// TIA Portal V16 export
// export: Created 2023-09-11T12:14:51.1549181Z, ExportSetting WithDefaults, DisplayName Totally Integrated Automation Portal, DisplayVersion V16 Update 6, DisplayName TIA Portal Version Control Interface, DisplayVersion V16 Update 2, DisplayName TIA Portal Openness, DisplayVersion V16 Update 6, DisplayName STEP 7 Professional, DisplayVersion V16 Update 6, DisplayName STEP 7 Safety, DisplayVersion V16, DisplayName WinCC Advanced, DisplayVersion V16 Update 6
ORGANIZATION_BLOCK "Cyclic interrupt"   // OB30, LAD, CyclicInterrupt
{ S7_Optimized_Access := 'TRUE' }
AUTHOR : RTecmer
VERSION : 0.1
// stored: AutoNumber true, IsIECCheckEnabled false, SetENOAutomatically false
   VAR_TEMP
      Temp_SV_Int : Int;
      PV_Temp : Real;
      Temp_1 : Real;
   END_VAR
   VAR_TEMP   // added for the SCL form of the ladder/FBD networks
      _w1 : Bool;
      _w2 : Bool;
   END_VAR
BEGIN

REGION Network 1: Wyłączenie wejścia pradowego w regulatorze PID
   // Przełączenie na Input PID  (wejście wartościci zadanej) wyłaczenie wejścia prądowego input_PER
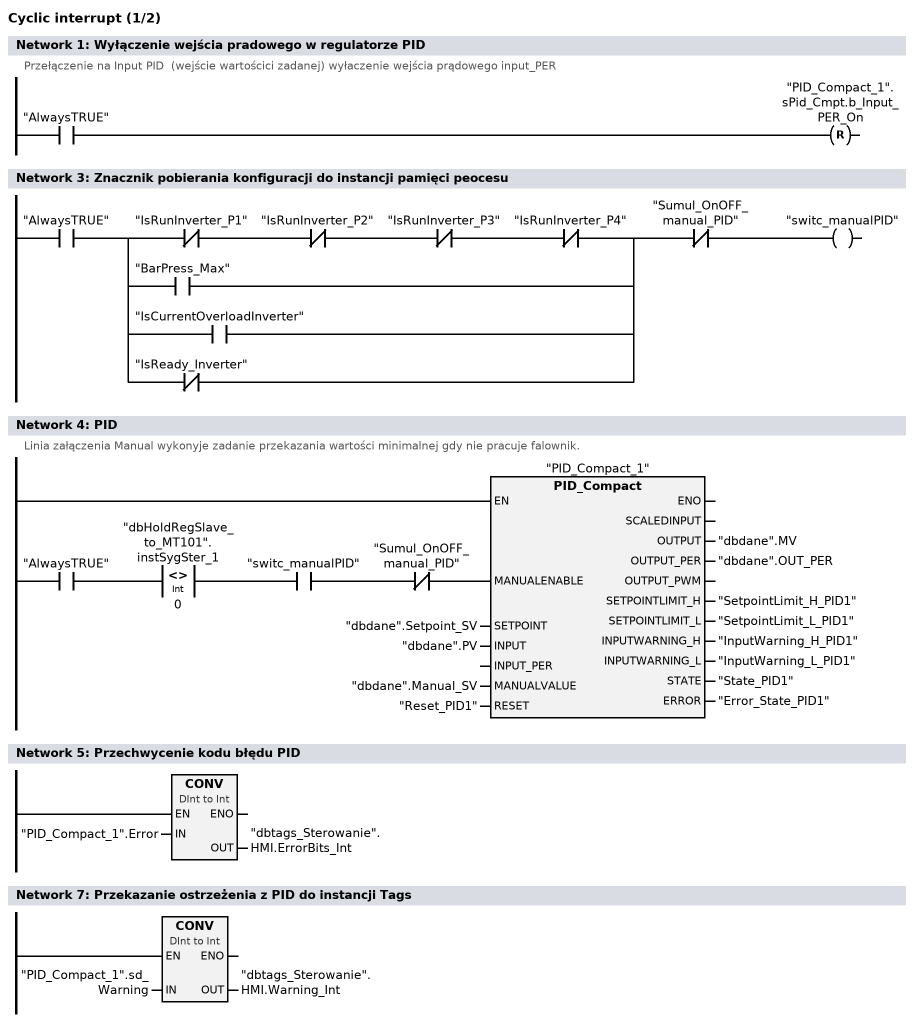
   RUNG wire#powerrail
      Contact( "AlwaysTRUE" )
      R_Coil( "PID_Compact_1".sPid_Cmpt.b_Input_PER_On )
   END_RUNG
   // the same network as SCL:
   IF "AlwaysTRUE" THEN "PID_Compact_1".sPid_Cmpt.b_Input_PER_On := FALSE; END_IF;
END_REGION

REGION Network 2: Skalowanie wartośc pressure oxygen
   // Przetwornik ciśnienia (0-1bar) 
   // !!!!!! Znienić po zamontowaniu właściwego !!!!!!! 
   // obecnie czujnik 10 bar
END_REGION

REGION Network 3: Znacznik pobierania konfiguracji do instancji pamięci peocesu
   RUNG wire#powerrail
      Contact( "AlwaysTRUE" )
      wire#w1
      I_Contact( "IsRunInverter_P1" )
      I_Contact( "IsRunInverter_P2" )
      I_Contact( "IsRunInverter_P3" )
      I_Contact( "IsRunInverter_P4" )
      wire#w2
      I_Contact( "Sumul_OnOFF_manual_PID" )
      Coil( "switc_manualPID" )
   END_RUNG
   RUNG wire#w1
      Contact( "BarPress_Max" )
   END_RUNG wire#w2
   RUNG wire#w1
      Contact( "IsCurrentOverloadInverter" )
   END_RUNG wire#w2
   RUNG wire#w1
      I_Contact( "IsReady_Inverter" )
   END_RUNG wire#w2
   // the same network as SCL:
   "switc_manualPID" := "AlwaysTRUE" AND ((NOT "IsRunInverter_P1" AND NOT "IsRunInverter_P2" AND NOT "IsRunInverter_P3" AND NOT "IsRunInverter_P4") OR "BarPress_Max" OR "IsCurrentOverloadInverter" OR NOT "IsReady_Inverter") AND NOT "Sumul_OnOFF_manual_PID";
END_REGION

REGION Network 4: PID
   // Linia załączenia Manual wykonyje zadanie przekazania wartości minimalnej gdy nie pracuje falownik.
   RUNG wire#powerrail
      "PID_Compact_1".PID_Compact(ManualEnable := wire#w1, Setpoint := "dbdane".Setpoint_SV, Input := "dbdane".PV, Input_PER :=, ManualValue := "dbdane".Manual_SV, Reset := "Reset_PID1", ScaledInput =>, Output => "dbdane".MV, Output_PER => "dbdane".OUT_PER, Output_PWM =>, SetpointLimit_H => "SetpointLimit_H_PID1", SetpointLimit_L => "SetpointLimit_L_PID1", InputWarning_H => "InputWarning_H_PID1", InputWarning_L => "InputWarning_L_PID1", State => "State_PID1", Error => "Error_State_PID1")
   END_RUNG
   RUNG wire#powerrail
      Contact( "AlwaysTRUE" )
      { S7_Templates := "SrcType := Int" } NE_Contact(in1 := "dbHoldRegSlave_to_MT101".instSygSter_1, in2 := 0)
      Contact( "switc_manualPID" )
      I_Contact( "Sumul_OnOFF_manual_PID" )
   END_RUNG wire#w1
   // the same network as SCL:
   "PID_Compact_1"(ManualEnable := "AlwaysTRUE" AND ("dbHoldRegSlave_to_MT101".instSygSter_1 <> 0) AND "switc_manualPID" AND NOT "Sumul_OnOFF_manual_PID",   // PID_Compact
                   Setpoint := "dbdane".Setpoint_SV,
                   Input := "dbdane".PV,
                   ManualValue := "dbdane".Manual_SV,
                   Reset := "Reset_PID1",
                   Output => "dbdane".MV,
                   Output_PER => "dbdane".OUT_PER,
                   SetpointLimit_H => "SetpointLimit_H_PID1",
                   SetpointLimit_L => "SetpointLimit_L_PID1",
                   InputWarning_H => "InputWarning_H_PID1",
                   InputWarning_L => "InputWarning_L_PID1",
                   State => "State_PID1",
                   Error => "Error_State_PID1");
END_REGION

REGION Network 5: Przechwycenie kodu błędu PID
   RUNG wire#powerrail
      { S7_Templates := "[SrcType := DInt, DestType := Int]"; S7_GenerateENO := "TRUE" } Convert(in := "PID_Compact_1".Error, out => "dbtags_Sterowanie".HMI.ErrorBits_Int)
   END_RUNG
   // the same network as SCL:
   "dbtags_Sterowanie".HMI.ErrorBits_Int := DINT_TO_INT("PID_Compact_1".Error);
END_REGION

REGION Network 7: Przekazanie ostrzeżenia z PID do instancji Tags
   RUNG wire#powerrail
      { S7_Templates := "[SrcType := DInt, DestType := Int]"; S7_GenerateENO := "TRUE" } Convert(in := "PID_Compact_1".sd_Warning, out => "dbtags_Sterowanie".HMI.Warning_Int)
   END_RUNG
   // the same network as SCL:
   "dbtags_Sterowanie".HMI.Warning_Int := DINT_TO_INT("PID_Compact_1".sd_Warning);
END_REGION

REGION Network 8: PID error reset
   // Reset PID od błędu
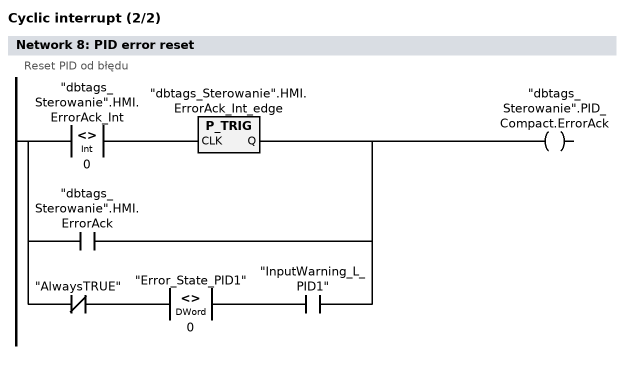
   RUNG wire#powerrail
      { S7_Templates := "SrcType := Int" } NE_Contact(in1 := "dbtags_Sterowanie".HMI.ErrorAck_Int, in2 := 0)
      P_Trig( "dbtags_Sterowanie".HMI.ErrorAck_Int_edge )
      wire#w1
      Coil( "dbtags_Sterowanie".PID_Compact.ErrorAck )
   END_RUNG
   RUNG wire#powerrail
      Contact( "dbtags_Sterowanie".HMI.ErrorAck )
   END_RUNG wire#w1
   RUNG wire#powerrail
      I_Contact( "AlwaysTRUE" )
      { S7_Templates := "SrcType := DWord" } NE_Contact(in1 := "Error_State_PID1", in2 := 0)
      Contact( "InputWarning_L_PID1" )
   END_RUNG wire#w1
   // the same network as SCL:
   #_w1 := "dbtags_Sterowanie".HMI.ErrorAck_Int <> 0;
   #_w2 := #_w1 AND NOT "dbtags_Sterowanie".HMI.ErrorAck_Int_edge;   // rising edge
   "dbtags_Sterowanie".HMI.ErrorAck_Int_edge := #_w1;
   "dbtags_Sterowanie".PID_Compact.ErrorAck := #_w2 OR "dbtags_Sterowanie".HMI.ErrorAck OR (NOT "AlwaysTRUE" AND ("Error_State_PID1" <> 0) AND "InputWarning_L_PID1");
END_REGION
END_ORGANIZATION_BLOCK
